// TwinCAT 3 PLC project Application
// ProgramVersion: 3.1.4024.0
// libraries:
//   Tc2_Standard, * (Beckhoff Automation GmbH)
//   Tc2_System, * (Beckhoff Automation GmbH)
//   Tc3_Module, * (Beckhoff Automation GmbH)
//   VisuDialogs, * (System)
//   VisuSymbols,3.5.10.0,System
// project tree:
//   DUTs/01_Schnittstellen/ I_HKSystem.TcIO (not stored), I_Magnetventil.TcIO (not stored), I_Motor1R.TcIO (not stored), I_Motor2R.TcIO, I_Sensor.TcIO
//   DUTs/02_Strukturen/ RezeptControlWord.TcDUT, RezeptStatusWord.TcDUT, SekControlWord.TcDUT, SystemStatusWord.TcDUT (not stored)
//   / GlobalTextList.TcGTLO, PlcTask.TcTTO, Visualisierungsmanager.TcVMO (not stored)
//   GVLs/01_OPC_UA/ GVL_OPC_UA.TcGVL
//   GVLs/ GVL.TcGVL
//   POUs/01_Objektklassen/ FB_A_HKSystem.TcPOU, FB_A_Magnetventil.TcPOU, FB_A_Motor1R.TcPOU, FB_A_Motor2R.TcPOU, FB_S_Sensor.TcPOU (not stored)
//   POUs/02_Anlage/01_Hilfsbausteine/ FB_Modus.TcPOU (not stored)
//   POUs/02_Anlage/ Reaktoreinheit.TcPOU
//   POUs/03_Grundfuntkionen/01_Vererbung/ FB_Basis.TcPOU
//   POUs/03_Grundfuntkionen/ GF_Befuellen.TcPOU, GF_Entleeren.TcPOU, GF_Pumpen.TcPOU, GF_Zirkulieren.TcPOU, GF_Ruehren.TcPOU, GF_Warten.TcPOU
//   POUs/04_Kommunikation/01_Hilfsfunktionsblock/ FB_Leitungswahl.TcPOU (not stored)
//   POUs/04_Kommunikation/ FB_Auswertung.TcPOU, Kommunikation.TcPOU
//   POUs/05_Simulation/ FB_SIM_Fuellstand.TcPOU
//   POUs/ MAIN.TcPOU
// real-time tasks:
//   TASK PlcTask: cycle T#10ms, priority 20, ADS port 350
//   TASK VISU_TASK: cycle T#200000us, priority 30, ADS port 351

CONFIGURATION Application
    RESOURCE PLC ON TwinCAT3
        TASK PlcTask(INTERVAL := T#10ms, PRIORITY := 20);
        PROGRAM MAIN WITH PlcTask : MAIN;
    END_RESOURCE
END_CONFIGURATION

// ---- DUTs/02_Strukturen/RezeptControlWord.TcDUT
TYPE RezeptControlWord :
STRUCT
	PowerOn			:BOOL;			// Einschalten von Reaktoreinheit
	SekReakt		:INT;			// Definierter sekundär-Reaktor
	Leitung			:INT;			// Definiert welche Leitung verwendet wird
	Temp			:REAL;			// Definierte Temperatur für Heiz- / Kühlprozess
	Enlteermenge	:REAL;			// Zu entleerende Menge
	Pumpmenge		:REAL;			// Zu pumpende Menge
	Haltedauer		:INT;			// Wie lange soll TEmperatur gehalten werden
	Ruehrdauer		:INT;			// Wie lange soll gerührt werden 
	Wartedauer		:INT;			// Wie lange soll gerührt werden
	Zirkulierdauer	:INT;			// Wie lange soll zirkuliert werden
END_STRUCT
END_TYPE

// ---- DUTs/02_Strukturen/RezeptStatusWord.TcDUT
TYPE RezeptStatusWord :
STRUCT
	SysReady		:BOOL;		// System ist bereit für Kommunikation
	SysActiv		:BOOL;		// System ist eingeschalten
	ReactReady		:BOOL;		// Primärreaktor ist bereit für den Prozess
	ReactActiv		:BOOL;		// Primärreaktor führt Prozess aus
	GF1Activ		:BOOL;		// Heiz- / Kühlprozess läuft
	GF2Activ		:BOOL;		// Entleerprozess läuft
	GF3Activ		:BOOL;		// Pumpprozess läuft
	GF4Activ		:BOOL;		// Halteprozess läuft
	GF5Activ		:BOOL;		// Rührprozess läuft
	GF6Activ		:BOOL;		// Warteprozess läuft
	GF7Activ		:BOOL;		// Auffüllprozess läuft
	GF8Activ		:BOOL;		// Zirkulierprozess läuft
END_STRUCT
END_TYPE

// ---- DUTs/02_Strukturen/SekControlWord.TcDUT
TYPE SekControlWord :
STRUCT
	// Das SekControlWord startet den Befüllprozess beim Sekundärreaktor (Empfänger)	
	R1				:BOOL;
	R2				:BOOL;
	R3				:BOOL;
	R4				:BOOL;
	R5				:BOOL;
	R6				:BOOL;
	R7				:BOOL;
END_STRUCT
END_TYPE

// ---- GVLs/01_OPC_UA/GVL_OPC_UA.TcGVL
{attribute 'qualified_only'}
VAR_GLOBAL
	// Rezept-Controlword
	{attribute 'OPC.UA.DA' := '1'}
	{attribute 'OPC.UA.DA.StructuredType' := '1'}
	CW			:RezeptControlWord;
	
	// Rezept-Statusword
	{attribute 'OPC.UA.DA' := '1'}
	{attribute 'OPC.UA.DA.Access' := '1'}
	{attribute 'OPC.UA.DA.StructuredType' := '1'}
	SW			:RezeptStatusWord;
	
	// System-Statusword
	{attribute 'OPC.UA.DA' := '1'}
	{attribute 'OPC.UA.DA.StructuredType' := '1'}
	SysSW		:SystemStatusWord;
	
	// Sekundärreaktor-Controlword
	{attribute 'OPC.UA.DA' := '1'}
	{attribute 'OPC.UA.DA.StructuredType' := '1'}
	SekCW		:SekControlWord;
END_VAR

// ---- GVLs/GVL.TcGVL
{attribute 'qualified_only'}
VAR_GLOBAL
	
	// Systemzustand
	SysState			:INT;		// 0 = Grundfunktion nicht aktive | 1 = Grundfunktion aktive

	// Bedienparameter
	Bedien_Power		:BOOL;
	Bedien_Reset		:BOOL;
	
	// Debug-Variablen: 
	Debug_Verbunden		:BOOL := TRUE;
	Debug_Start			:BOOL := TRUE;
	Debug_SekStart		:BOOL;
	
	// Simulationsvariablen 
	Sim_StandSignal		:INT;
	Sim_Fuellen			:BOOL;

END_VAR

// ---- DUTs/01_Schnittstellen/I_Motor2R.TcIO
INTERFACE I_Motor2R

METHOD M_A_BWD : BOOL
VAR_INPUT
END_VAR
END_METHOD

METHOD M_A_FWD : BOOL
VAR_INPUT
END_VAR
END_METHOD

METHOD M_A_START : BOOL
VAR_INPUT
END_VAR
END_METHOD

METHOD M_A_STOP : BOOL
VAR_INPUT
END_VAR
END_METHOD

METHOD M_M_BWD : BOOL
VAR_INPUT
END_VAR
END_METHOD

METHOD M_M_FWD : BOOL
VAR_INPUT
END_VAR
END_METHOD

METHOD M_M_START : BOOL
VAR_INPUT
END_VAR
END_METHOD

METHOD M_M_STOP : BOOL
VAR_INPUT
END_VAR
END_METHOD

PROPERTY P_Laufzeit : TIME
GET
END_GET
END_PROPERTY

PROPERTY P_MaxDrz : INT
SET
END_SET
END_PROPERTY

PROPERTY P_Status : INT
GET
END_GET
END_PROPERTY

END_INTERFACE

// ---- DUTs/01_Schnittstellen/I_Sensor.TcIO
INTERFACE I_Sensor

PROPERTY P_GrenzeOben : BOOL
GET
END_GET
END_PROPERTY

PROPERTY P_GrenzeUnten : BOOL
GET
END_GET
END_PROPERTY

PROPERTY P_Messwert : REAL
GET
END_GET
END_PROPERTY

END_INTERFACE

// ---- POUs/MAIN.TcPOU
PROGRAM MAIN
VAR
	Simulation		:FB_Sim_Fuellstand;
	Sim_ON			:BOOL := TRUE;
END_VAR

VAR_INPUT
	// Statusword
	
	// Sonstiges
END_VAR

// Starten der Reaktoreinheit
Reaktoreinheit();

// Starten der Auswertung der Kommunikationsschnittstelle
Kommunikation();

// Simulation starten
IF Sim_ON THEN
	Simulation(I_Fuellen := GVL.Sim_Fuellen,
			   O_SensorSignal => GVL.Sim_StandSignal);
			   
	Reaktoreinheit.F1.I_iSignal := GVL.Sim_StandSignal;
END_IF

END_PROGRAM

// ---- POUs/05_Simulation/FB_SIM_Fuellstand.TcPOU
FUNCTION_BLOCK FB_SIM_Fuellstand
VAR_INPUT
	I_Fuellen			:BOOL;
END_VAR

VAR_OUTPUT
	O_SensorSignal		:INT;
END_VAR
	
VAR
	V_Delay				:TON;
	V_TimeStatus		:BOOL;
END_VAR

// Timer instanziieren
V_Delay(IN := V_TimeStatus, PT := T#1S);	

IF I_Fuellen THEN
	// Grundwert definieren
	O_SensorSignal := 0;
	
	// Timer starten
	V_TimeStatus := TRUE;
	
	// Reaktor füllen
	IF V_Delay.Q THEN
		V_TimeStatus := FALSE;
		O_SensorSignal := O_SensorSignal + (27648/100);
	END_IF
END_IF

END_FUNCTION_BLOCK

// ---- POUs/02_Anlage/Reaktoreinheit.TcPOU
PROGRAM Reaktoreinheit
VAR
	// Allgemeine Instanziierungen
	Mode					:FB_Modus;
	
	// Instanziierung der Aktoren
	YSE1, YSE2				:FB_A_Magnetventil;
	YSA1, YSA2, YSA3		:FB_A_Magnetventil;
	YSP1, YSP2, YSP3		:FB_A_Magnetventil;
	
	NC1						:FB_A_Motor1R;
	
	PS1						:FB_A_Motor2R;
	
	HKP1					:FB_A_HKSystem;
END_VAR

VAR_INPUT
		// Instanziierung der Sensoren
	T1						:FB_S_Sensor;
	F1						:FB_S_Sensor;
END_VAR

YSE1(I_iModus := Mode.O_iModus); // FB_A_Magnetventil
YSP3(I_iModus := Mode.O_iModus); // FB_A_Magnetventil
F1(I_rHigh := 27648, I_rLow := 0, I_rMax := 100, I_rMin := 0); // FB_S_Sensor
Mode(I_bPower := GVL.Bedien_Power); // FB_Modus
YSA3(I_iModus := Mode.O_iModus); // FB_A_Magnetventil
HKP1(
    I_bVerbunden := GVL.Debug_Verbunden,
    I_iModus := Mode.O_iModus,
    I_iTemp := T1.P_Messwert,
    I_bReset := GVL.Bedien_Reset); // FB_A_HKSystem
YSA2(I_iModus := Mode.O_iModus); // FB_A_Magnetventil
YSP2(I_iModus := Mode.O_iModus); // FB_A_Magnetventil
PS1(
    I_bVerbunden := GVL.Debug_Verbunden,
    I_iModus := Mode.O_iModus,
    I_bReset := GVL.Bedien_Reset,
    I_iGeschw := 100); // FB_A_Motor2R
NC1(I_iModus := Mode.O_iModus, I_bReset := GVL.Bedien_Reset, I_iGeschw := 100); // FB_A_Motor1R
YSE2(I_iModus := Mode.O_iModus); // FB_A_Magnetventil
YSA1(I_iModus := Mode.O_iModus); // FB_A_Magnetventil
YSP1(I_iModus := Mode.O_iModus); // FB_A_Magnetventil
T1(I_rHigh := 27648, I_rLow := 0, I_rMax := 100, I_rMin := 0); // FB_S_Sensor

END_PROGRAM

// ---- POUs/01_Objektklassen/FB_A_Magnetventil.TcPOU
FUNCTION_BLOCK FB_A_Magnetventil IMPLEMENTS I_Magnetventil
VAR_INPUT
	I_iModus			:INT;		// Zustand des Systems (z.B. 0 = AUS | 1 = MAN | 2 = AUTO)
	I_bVerriegeln		:BOOL;		// Verriegelte Elemente sind nicht ansteuerbar
END_VAR

VAR_OUTPUT
	O_bAktivieren		:BOOL;		// Ventil wird geöffnet / geschlossen
	O_bStoerung			:BOOL;		// Befindet sich das Element in einem Error
	O_iStoerungID		:INT;		// Anzeigen von Störung über eine INT-Variable
END_VAR

VAR
END_VAR

// Verriegeln des Systems (Element geht in definierten Zustand) -> Ventil wird geschlossen
IF I_bVerriegeln THEN
	O_bAktivieren := FALSE;
END_IF

METHOD M_A_OEFFNEN : BOOL
VAR_INPUT
END_VAR
// EBENE 1: Verriegelung
IF NOT I_bVerriegeln THEN	
	// EBEN 2: AUTO-Modus
		IF I_iModus = 2 THEN
			O_bAktivieren := TRUE;
		END_IF
END_IF

M_A_OEFFNEN := O_bAktivieren;
END_METHOD

METHOD M_A_SCHLIESSEN : BOOL
VAR_INPUT
END_VAR
IF I_iModus = 2 THEN
	O_bAktivieren := FALSE;
END_IF

M_A_SCHLIESSEN := NOT O_bAktivieren;
END_METHOD

METHOD M_M_OEFFNEN : BOOL
VAR_INPUT
END_VAR
// EBENE 1: Verriegelung
IF NOT I_bVerriegeln THEN	
	// EBEN 2: MAN-Modus
		IF I_iModus = 1 THEN
			O_bAktivieren := TRUE;
		END_IF
END_IF

M_M_OEFFNEN := O_bAktivieren;
END_METHOD

METHOD M_M_SCHLIESSEN : BOOL
VAR_INPUT
END_VAR
IF I_iModus = 1 THEN
	O_bAktivieren := FALSE;
END_IF

M_M_SCHLIESSEN := NOT O_bAktivieren;
END_METHOD

PROPERTY P_Status : INT
GET
IF O_bAktivieren THEN
	P_Status := 1;
ELSE
	P_Status := 0;
END_IF

IF I_bVerriegeln THEN
	P_Status := 10;
END_IF
END_GET
END_PROPERTY

END_FUNCTION_BLOCK

// ---- POUs/01_Objektklassen/FB_A_Motor1R.TcPOU
FUNCTION_BLOCK FB_A_Motor1R IMPLEMENTS I_Motor1R
VAR_INPUT
	I_iModus			:INT;		// Zustand des Systems (z.B. 0 = AUS | 1 = MAN | 2 = AUTO | 3 = Error)
	I_bVerriegeln		:BOOL;		// Verriegelte Elemente sind nicht ansteuerbar
	I_bReset			:BOOL;		// Zustand des Baustein wird zurückgesetzt 
	I_iGeschw			:INT;		// Angabe über Soll-Geschwindigkeit
END_VAR

VAR_OUTPUT
	O_bPower			:BOOL;		// Relais wird geschalten um FU mit Spannung zu versorgen
	O_iDrz				:INT;		// Ausgabe der Drehzahl für den Motor (Umrechnen von Spannung zu Drz)
	O_bStoerung			:BOOL;		// Befindet sich das Element in einem Error
	O_iStoerungID		:INT;		// Anzeigen von Störung über eine INT-Variable
END_VAR

VAR
	V_DrzMax		:INT;		// Variable für internes handling der Eigenschaft 
	V_Zeit			:TIME;		// Variable für internes handling der Eigenschaft 
	V_Status		:INT;		// Variable für internes handling der Eigenschaft 
	
	V_Timer			:TON;		// Runtime des Bausteins ermitteln
	
END_VAR

// Setzen der internen Variablen
P_MaxDrz := V_DrzMax;
V_Zeit := P_Laufzeit;
V_Status := P_Status;

// Reset des Bausteins
IF I_bReset THEN
	O_bStoerung := FALSE;
	O_iStoerungID := 0;
END_IF

// Verriegeln des Systems (Element geht in definierten Zustand) -> Motor wird gestoppt und ausgeschalten
IF I_bVerriegeln THEN
	O_iDrz := 0;
	O_bPower := FALSE;
END_IF

METHOD M_A_AN : BOOL
VAR_INPUT
END_VAR
// EBENE 1: Verriegelung
IF NOT I_bVerriegeln THEN	
	// EBEN 2: AUTO-Modus
		IF I_iModus = 2 THEN
			O_bPower := TRUE;
		END_IF
ELSE 
	O_bPower := FALSE;
END_IF

M_A_AN := O_bPower;
END_METHOD

METHOD M_A_AUS : BOOL
VAR_INPUT
END_VAR
IF I_iModus = 2 THEN
	O_bPower := FALSE;
	O_iDrz := 0;
END_IF

M_A_AUS := NOT O_bPower;
END_METHOD

METHOD M_A_START : BOOL
VAR_INPUT
END_VAR
// EBENE 1: Verriegelung
IF NOT I_bVerriegeln THEN

	// EBENE 2: Check der Drehzzahl
	IF I_iGeschw <= V_DrzMax THEN
		
		// Ebene 3: AUTO-Modus
		IF I_iModus = 2 THEN
			
			// EBENE 4: System muss AN sein
			IF O_bPower THEN
				O_iDrz := I_iGeschw;
				
			ELSE 	// Error: System ist nicht eingeschalten
				O_bStoerung := 1;
				O_iStoerungID := 11; 
		END_IF
		
	ELSE	// Error: Geschwindigkeit überschreitet die MaxDrz
		O_bStoerung := 1;
		O_iStoerungID := 12;
		END_IF		
	END_IF
END_IF

IF O_iDrz = I_iGeschw THEN
	M_A_START := TRUE;
ELSE
	M_A_START := FALSE;
END_IF
END_METHOD

METHOD M_A_STOP : BOOL
VAR_INPUT
END_VAR
// EBENE 1: Verriegelung
IF NOT I_bVerriegeln THEN
	O_iDrz := 0;
END_IF

IF O_iDrz = 0 THEN
	M_A_STOP := TRUE;
ELSE
	M_A_STOP := FALSE;
END_IF
END_METHOD

METHOD M_M_AN : BOOL
VAR_INPUT
END_VAR
// EBENE 1: Verriegelung
IF NOT I_bVerriegeln THEN	
	// EBEN 2: MAN-Modus
		IF I_iModus = 1 THEN
			O_bPower := TRUE;
		END_IF
ELSE 
	O_bPower := FALSE;
END_IF

M_M_AN := O_bPower;
END_METHOD

METHOD M_M_AUS : BOOL
VAR_INPUT
END_VAR
IF I_iModus = 1 THEN
	O_bPower := FALSE;
	O_iDrz := 0;
END_IF

M_M_AUS := NOT O_bPower;
END_METHOD

METHOD M_M_START : BOOL
VAR_INPUT
END_VAR
// EBENE 1: Verriegelung
IF NOT I_bVerriegeln THEN

	// EBENE 2: Check der Drehzzahl
	IF I_iGeschw <= V_DrzMax THEN
		
		// EBENE 3: MAN-Modus
		IF I_iModus = 1 THEN
			
			// EBENE 4: System muss AN sein
			IF O_bPower THEN
				O_iDrz := I_iGeschw;
				
			ELSE 	// Error: System ist nicht eingeschalten
				O_bStoerung := 1;
			O_iStoerungID := 11;
			END_IF
		END_IF
		
	ELSE	// Error: Geschwindigkeit überschreitet die MaxDrz
		O_bStoerung := 1;
		O_iStoerungID := 12;
	END_IF		
END_IF

IF O_iDrz = I_iGeschw THEN
	M_M_START := TRUE;
ELSE
	M_M_START := FALSE;
END_IF
END_METHOD

METHOD M_M_STOP : BOOL
VAR_INPUT
END_VAR
// EBENE 1: Verriegelung
IF NOT I_bVerriegeln THEN
	O_iDrz := 0;
END_IF

IF O_iDrz = 0 THEN
	M_M_STOP := TRUE;
ELSE
	M_M_STOP := FALSE;
END_IF
END_METHOD

PROPERTY PUBLIC P_Laufzeit : TIME
GET
IF O_iDrz > 0 THEN
	V_Timer(IN := TRUE, PT := T#100H);
END_IF

IF O_iDrz = 0 THEN
	V_Timer(IN := FALSE);
END_IF 
P_Laufzeit := V_Timer.ET;
END_GET
END_PROPERTY

PROPERTY PUBLIC P_MaxDrz : INT
SET
END_SET
END_PROPERTY

PROPERTY PUBLIC P_Status : INT
GET
IF O_bPower THEN
	P_Status := 1;
ELSE
	P_Status := 0;
END_IF

IF O_iDrz > 0 AND O_bPower THEN
	P_Status := 2;
END_IF

IF I_bVerriegeln THEN
	P_Status := 10;
END_IF
END_GET
END_PROPERTY

END_FUNCTION_BLOCK

// ---- POUs/01_Objektklassen/FB_A_Motor2R.TcPOU
FUNCTION_BLOCK FB_A_Motor2R IMPLEMENTS I_Motor2R
VAR_INPUT
	I_bVerbunden		:BOOL;		// Angabe ob Pumpe angeschlossen ist
	I_iModus			:INT;		// Zustand des Systems (z.B. 0 = AUS | 1 = MAN | 2 = AUTO)
	I_bVerriegeln		:BOOL;		// Verriegelte Elemente sind nicht ansteuerbar
	I_bReset			:BOOL;		// Zustand des Baustein wird zurückgesetzt 
	I_iGeschw			:INT;		// Angabe über Soll-Geschwindigkeit
END_VAR

VAR_OUTPUT
	
	O_iDrz				:INT;		// Ausgabe der Drehzahl für den Motor
	O_bRichtung			:BOOL;		// Ausgabe der Drehrichtung
	O_bStoerung			:BOOL;		// Befindet sich das Element in einem Error
	O_iStoerungID		:INT;		// Anzeigen von Störung über eine INT-Variable
END_VAR

VAR
	V_DrzMax		:INT;		// Variable für internes handling der Eigenschaft 
	V_Zeit			:TIME;		// Variable für internes handling der Eigenschaft 
	V_Zustand		:INT;		// Variable für internes handling der Eigenschaft

	V_Timer			:TON;		// Runtime des Bausteins ermitteln 
END_VAR

// Setzen der internen Variablen
P_MaxDrz := V_DrzMax;
V_Zeit := P_Laufzeit;
V_Zustand := P_Status;

// Reset des Bausteins
IF I_bReset THEN
	O_bStoerung := FALSE;
	O_iStoerungID := 0;
END_IF

// Verriegeln des Systems (Element geht in definierten Zustand) -> Motor wird hält an 
IF I_bVerriegeln THEN
	O_iDrz := 0;
	O_bRichtung := FALSE;
END_IF

METHOD M_A_BWD : BOOL
VAR_INPUT
END_VAR
// EBENE 1: Verriegelung
IF NOT I_bVerriegeln THEN	
	// EBENE 2: AUTO-Modus
		IF I_iModus = 2 THEN
			// EBENE 3: System muss angeschlossen sein
			IF I_bVerbunden THEN
				O_bRichtung := TRUE;
			ELSE 	// Error: System ist nicht angeschlossen
				O_bStoerung := 1;
				O_iStoerungID := 03;
			END_IF
		END_IF
END_IF

M_A_BWD := O_bRichtung;
END_METHOD

METHOD M_A_FWD : BOOL
VAR_INPUT
END_VAR
// EBENE 1: Verriegelung
IF NOT I_bVerriegeln THEN	
	// EBENE 2: AUTO-Modus
		IF I_iModus = 2 THEN
			// EBENE 3: System muss angeschlossen sein
			IF I_bVerbunden THEN
				O_bRichtung := FALSE;
			ELSE 	// Error: System ist nicht angeschlossen
				O_bStoerung := 1;
				O_iStoerungID := 03;
			END_IF
		END_IF
END_IF

M_A_FWD := NOT O_bRichtung;
END_METHOD

METHOD M_A_START : BOOL
VAR_INPUT
END_VAR
// EBENE 1: Verriegelung
IF NOT I_bVerriegeln THEN

	// EBENE 2: Check der Drehzzahl
	IF I_iGeschw <= V_DrzMax THEN
		
		// EBENE 3: AUTO-Modus
		IF I_iModus = 2 THEN
			
			// EBENE 4: System muss angeschlossen sein
			IF I_bVerbunden THEN
				O_iDrz := I_iGeschw;
				
			ELSE 	// Error: System ist nicht angeschlossen
				O_bStoerung := 1;
				O_iStoerungID := 03;
			END_IF
		END_IF
		
	ELSE	// Error: Geschwindigkeit überschreitet die MaxDrz
		O_bStoerung := 1;
		O_iStoerungID := 01;
	END_IF		
END_IF

IF O_iDrz = I_iGeschw THEN
	M_A_START := TRUE;
END_IF
END_METHOD

METHOD M_A_STOP : BOOL
VAR_INPUT
END_VAR
// EBENE 1: Verriegelung
IF NOT I_bVerriegeln THEN
	O_iDrz := 0;
END_IF

IF O_iDrz = 0 THEN
	M_A_STOP := TRUE;
END_IF
END_METHOD

METHOD M_M_BWD : BOOL
VAR_INPUT
END_VAR
// EBENE 1: Verriegelung
IF NOT I_bVerriegeln THEN	
	// EBENE 2: MAN-Modus
		IF I_iModus = 1 THEN
			// EBENE 3: System muss angeschlossen sein
			IF I_bVerbunden THEN
				O_bRichtung := TRUE;
			ELSE 	// Error: System ist nicht angeschlossen
				O_bStoerung := 1;
				O_iStoerungID := 03;
			END_IF
		END_IF
END_IF

M_M_BWD := O_bRichtung;
END_METHOD

METHOD M_M_FWD : BOOL
VAR_INPUT
END_VAR
// EBENE 1: Verriegelung
IF NOT I_bVerriegeln THEN	
	// EBENE 2: MAN-Modus
		IF I_iModus = 1 THEN
			// EBENE 3: System muss angeschlossen sein
			IF I_bVerbunden THEN
				O_bRichtung := FALSE;
			ELSE 	// Error: System ist nicht angeschlossen
				O_bStoerung := 1;
				O_iStoerungID := 03;
			END_IF
		END_IF
END_IF

M_M_FWD := NOT O_bRichtung;
END_METHOD

METHOD M_M_START : BOOL
VAR_INPUT
END_VAR
// EBENE 1: Verriegelung
IF NOT I_bVerriegeln THEN

	// EBENE 2: Check der Drehzzahl
	IF I_iGeschw <= V_DrzMax THEN
		
		// EBENE 3: MAN-Modus
		IF I_iModus = 1 THEN
			
			// EBENE 4: System muss angeschlossen sein
			IF I_bVerbunden THEN
				O_iDrz := I_iGeschw;
				
			ELSE 	// Error: System ist nicht angeschlossen
				O_bStoerung := 1;
				O_iStoerungID := 03;
			END_IF
		END_IF
		
	ELSE	// Error: Geschwindigkeit überschreitet die MaxDrz
		O_bStoerung := 1;
		O_iStoerungID := 01;
	END_IF		
END_IF

IF O_iDrz = I_iGeschw THEN
	M_M_START := TRUE;
END_IF
END_METHOD

METHOD M_M_STOP : BOOL
VAR_INPUT
END_VAR
// EBENE 1: Verriegelung
IF NOT I_bVerriegeln THEN
	O_iDrz := 0;
END_IF

IF O_iDrz = 0 THEN
	M_M_STOP := TRUE;
END_IF
END_METHOD

PROPERTY PUBLIC P_Laufzeit : TIME
GET
IF O_iDrz > 0 THEN
	V_Timer(IN := TRUE, PT := T#100H);
END_IF

IF O_iDrz = 0 THEN
	V_Timer(IN := FALSE);
END_IF 
P_Laufzeit := V_Timer.ET;
END_GET
END_PROPERTY

PROPERTY PUBLIC P_MaxDrz : INT
SET
END_SET
END_PROPERTY

PROPERTY PUBLIC P_Status : INT
GET
IF I_bVerbunden THEN
	P_Status := 1;
END_IF

IF I_bVerriegeln THEN
	P_Status := 10;
END_IF

IF O_iDrz > 0	THEN
	P_Status := 2;
END_IF
END_GET
END_PROPERTY

END_FUNCTION_BLOCK

// ---- POUs/01_Objektklassen/FB_A_HKSystem.TcPOU
FUNCTION_BLOCK FB_A_HKSystem IMPLEMENTS I_HKSystem
VAR_INPUT
	I_bVerbunden	:BOOL;		// Angabe ob HK-System angeschlossen ist
	I_iModus		:INT;		// Zustand des Systems (z.B. 0 = AUS | 1 = MAN | 2 = AUTO)
	I_iTemp			:REAL;		// Aktuelle Temperatur um Heizmodus auszuwählen und zu stoppen
	I_bVerriegeln	:BOOL;		// Verriegelte Elemente sind nicht ansteuerbar
	I_bReset		:BOOL;		// Zustand des Baustein wird zurückgesetzt 
END_VAR

VAR_OUTPUT
	O_bPumpen		:BOOL;		// Pumpe des HK-Systems wird betrieben
	O_bKuehlen		:BOOL;		// HK-System heizt das Medium auf
	O_bHeizen		:BOOL;		// HK-System kühlt das Medium ab
	O_bStoerung		:BOOL;		// Befindet sich das Element in einem Error
	O_iStoerungID	:INT;		// Anzeigen von Störung über eine INT-Variable
	
END_VAR
	
VAR
	V_DefTemp		:INT;		// Variable für internes handling der Eigenschaft 
	V_Zeit			:TIME;		// Variable für internes handling der Eigenschaft 
	V_Zustand		:INT;		// Variable für internes handling der Eigenschaft 
	
	V_Timer			:TON;		// Runtime des Bausteins ermitteln
END_VAR

// Setzen der internen Variablen
V_Zeit := P_Laufzeit;
V_Zustand := P_Zustand;

// Fehler durch Verbindungsabbruch
IF O_bPumpen OR O_bKuehlen OR O_bHeizen THEN
	IF NOT I_bVerbunden THEN
		O_bPumpen := FALSE;
		O_bKuehlen := FALSE;
		O_bHeizen := FALSE;
		
		O_bStoerung := TRUE;
		O_iStoerungID := 04;
	END_IF
END_IF

// Abbruch des Heiz-Kühlprozesses beim erreichen der Temp
IF O_bHeizen OR O_bKuehlen THEN 
	IF I_iTemp = V_DefTemp THEN
		O_bKuehlen := FALSE;
		O_bHeizen := FALSE;		
	END_IF
END_IF

// Reset des Bausteins
IF I_bReset THEN
	O_bStoerung := FALSE;
	O_iStoerungID := 0;
END_IF

METHOD M_A_HK_AN : BOOL
VAR_INPUT
END_VAR
// EBENE 1: Verriegelung
IF NOT I_bVerriegeln THEN	
	// EBENE 2: AUTO-Modus
		IF I_iModus = 2 THEN
			// EBENE 3: Ist Pumpe AN
				IF O_bPumpen THEN
				// EBENE 4: Heizen oder Kühlen
					IF V_DefTemp > I_iTemp THEN
						O_bKuehlen := FALSE;
						O_bHeizen := TRUE;
						
						M_A_HK_AN := O_bHeizen;
						
					ELSIF I_iTemp > V_DefTemp THEN 	
						O_bHeizen := FALSE;
						O_bKuehlen := TRUE;
						
						M_A_HK_AN := O_bKuehlen;
					END_IF
				ELSE // Error: System ist nicht eingeschalten
					O_bStoerung := 1;
					O_iStoerungID := 11; 
				END_IF
			END_IF
END_IF
END_METHOD

METHOD M_A_HK_AUS : BOOL
VAR_INPUT
END_VAR
// EBENE 1: Verriegelung
IF NOT I_bVerriegeln THEN
		O_bKuehlen := FALSE;
		O_bHeizen := FALSE;
END_IF

IF O_bKuehlen = FALSE THEN
	M_A_HK_AUS := TRUE;
END_IF
END_METHOD

METHOD M_A_PUMPE_AN : BOOL
VAR_INPUT
END_VAR
// EBENE 1: Verriegelung
IF NOT I_bVerriegeln THEN	
	// EBENE 2: AUTO-Modus
		IF I_iModus = 2 THEN
			// EBENE 3: System muss angeschlossen sein
			IF I_bVerbunden THEN
				O_bPumpen := TRUE;
			ELSE 	// Error: System ist nicht angeschlossen
				O_bStoerung := 1;
				O_iStoerungID := 03;
			END_IF
		END_IF
END_IF

M_A_PUMPE_AN := O_bPumpen;
END_METHOD

METHOD M_A_PUMPE_AUS : BOOL
VAR_INPUT
END_VAR
// EBENE 1: Verriegelung
IF NOT I_bVerriegeln THEN
	IF NOT O_bHeizen AND NOT O_bKuehlen THEN
		O_bPumpen := FALSE;
	ELSE
		O_bStoerung := TRUE;
		O_iStoerungID := 05;
	END_IF
END_IF

IF O_bPumpen = FALSE THEN
	M_A_PUMPE_AUS := TRUE;
END_IF
END_METHOD

METHOD M_M_HK_AN : BOOL
VAR_INPUT
END_VAR
// EBENE 1: Verriegelung
IF NOT I_bVerriegeln THEN	
	// EBENE 2: MAN-Modus
		IF I_iModus = 1 THEN
			// EBENE 3: Ist Pumpe AN
				IF O_bPumpen THEN
				// EBENE 4: Heizen oder Kühlen
					IF V_DefTemp > I_iTemp THEN
						O_bKuehlen := FALSE;
						O_bHeizen := TRUE;
						
						M_M_HK_AN := O_bHeizen;
						
					ELSIF I_iTemp > V_DefTemp THEN 	
						O_bHeizen := FALSE;
						O_bKuehlen := TRUE;
						
						M_M_HK_AN := O_bKuehlen;
					END_IF
				ELSE // Error: System ist nicht eingeschalten
				O_bStoerung := 1;
				O_iStoerungID := 11; 	
				END_IF
			END_IF
END_IF
END_METHOD

METHOD M_M_HK_AUS : BOOL
VAR_INPUT
END_VAR
// EBENE 1: Verriegelung
IF NOT I_bVerriegeln THEN
		O_bKuehlen := FALSE;
		O_bHeizen := FALSE;
END_IF

IF O_bKuehlen = FALSE THEN
	M_M_HK_AUS := TRUE;
END_IF
END_METHOD

METHOD M_M_PUMPE_AN : BOOL
VAR_INPUT
END_VAR
// EBENE 1: Verriegelung
IF NOT I_bVerriegeln THEN	
	// EBENE 2: MAN-Modus
		IF I_iModus = 1 THEN
			// EBENE 3: System muss angeschlossen sein
			IF I_bVerbunden THEN
				O_bPumpen := TRUE;
			ELSE 	// Error: System ist nicht angeschlossen
				O_bStoerung := 1;
				O_iStoerungID := 03;
			END_IF
		END_IF
END_IF

M_M_PUMPE_AN := O_bPumpen;
END_METHOD

METHOD M_M_PUMPE_AUS : BOOL
VAR_INPUT
END_VAR
// EBENE 1: Verriegelung
IF NOT I_bVerriegeln THEN
	IF NOT O_bHeizen AND NOT O_bKuehlen THEN
		O_bPumpen := FALSE;
	ELSE
		O_bStoerung := TRUE;
		O_iStoerungID := 05;
	END_IF
END_IF

IF O_bPumpen = FALSE THEN
	M_M_PUMPE_AUS := TRUE;
END_IF
END_METHOD

PROPERTY P_DefTemp : INT
SET
END_SET
END_PROPERTY

PROPERTY P_Laufzeit : TIME
GET
IF O_bKuehlen OR O_bHeizen THEN
	V_Timer(IN := TRUE, PT := T#100H);
ELSE
	V_Timer(IN := FALSE);
END_IF

P_Laufzeit := V_Timer.ET;
END_GET
END_PROPERTY

PROPERTY PUBLIC P_Zustand : INT
GET
END_GET
END_PROPERTY

END_FUNCTION_BLOCK

// ---- POUs/04_Kommunikation/Kommunikation.TcPOU
PROGRAM Kommunikation
VAR
	
	// Instanziierung der Auswertung:
	Auswertung		:FB_Auswertung;
	Mode			:FB_Modus;
	
	// Instanziierung der Grundfunktionen: 
	Entleeren		:GF_Entleeren;
	//Halten			:GF_Halten;
	Pumpen			:GF_Pumpen;
	Zirkulieren		:GF_Zirkulieren;
	Ruehren 		:GF_Ruehren;
	Warten			:GF_Warten;	
	Befuellen		:GF_Befuellen;	
	Leitung			:FB_Leitungswahl;

END_VAR

Auswertung(
    I_RNr := GVL_OPC_UA.CW.SekReakt,
    I_ControlWord := GVL_OPC_UA.CW,
    I_SystemStatusWord := GVL_OPC_UA.SysSW,
    I_SekCW := GVL_OPC_UA.SekCW); // FB_Auswertung
GVL_OPC_UA.SW := Auswertung.O_StatusWord;
GVL.Bedien_Power := Auswertung.O_SystemON;

END_PROGRAM

// ---- POUs/04_Kommunikation/FB_Auswertung.TcPOU
FUNCTION_BLOCK FB_Auswertung
VAR_INPUT
	I_Manuel			:BOOL;	
	I_RNr				:INT;				// Reaktornummer für korrekte Zuweisung von SystemStatusWord		
	I_ControlWord		:RezeptControlWord;
	I_SystemStatusWord	:SystemStatusWord;
	I_SekCW				:SekControlWord;
END_VAR
VAR_OUTPUT
	O_StatusWord		:RezeptStatusWord; 
	O_SystemON			:BOOL;
END_VAR
VAR
	V_Status			:INT;						// Variable für Case-Switch
	V_Aktiv				:BOOL;						// System ist aktiv
	V_GF_Switch			:INT;						// Definiert welche GF durchgegührt werden soll	
	V_SekRe				:BOOL;						// Wird aktiviert falls Reaktor als Sekundärreaktor eingesetzt wird
	V_SekReady			:BOOL;
	V_SekActiv			:BOOL;
END_VAR

// Befindet sich System in Manuel-Modus
IF I_Manuel THEN
	V_Status := 0;
END_IF  

// System befindet sich im Automatik-Modus, aber ist noch nicht aktiv
IF NOT I_Manuel AND NOT V_Aktiv THEN
	V_Status := 1;
END_IF

// Auswertung des SystemStatusWords 
CASE I_RNr OF 
	1:	V_SekReady := I_SystemStatusWord.R1_Ready;
		V_SekActiv := I_SystemStatusWord.R1_Activ;
	
	2:	V_SekReady := I_SystemStatusWord.R2_Ready;
		V_SekActiv := I_SystemStatusWord.R2_Activ;
	
	3:	V_SekReady := I_SystemStatusWord.R3_Ready;
		V_SekActiv := I_SystemStatusWord.R3_Activ;
	
	4:	V_SekReady := I_SystemStatusWord.R4_Ready;
		V_SekActiv := I_SystemStatusWord.R4_Activ;
		
	5:	V_SekReady := I_SystemStatusWord.R5_Ready;
		V_SekActiv := I_SystemStatusWord.R5_Activ;
	
	6:	V_SekReady := I_SystemStatusWord.R6_Ready;
		V_SekActiv := I_SystemStatusWord.R6_Activ;
	
	7:	V_SekReady := I_SystemStatusWord.R7_Ready;
		V_SekActiv := I_SystemStatusWord.R7_Activ;
END_CASE

CASE V_Status OF
	0: // System im Manuel-Modus
		O_StatusWord.SysReady := FALSE;
		
	//==================================================================================================
	1: // Auswerten von Controlwords bezüglich Systemstart
		// System ist Ready für Communikation
		O_StatusWord.SysReady := TRUE;
		
		// Falls Power eingeschalten wird und das System noch nicht Ein ist, wird System Aktiviert
		IF I_ControlWord.PowerOn AND NOT O_SystemON THEN
			V_Aktiv := TRUE;
			V_Status := 2;
		END_IF
		
		// Auswertung von Sekundärreaktor-Controlword bezüglich Empfänger-Prozes 
		CASE I_RNr OF 
			1: V_SekRe := I_SekCW.R1;
			2: V_SekRe := I_SekCW.R2;
			3: V_SekRe := I_SekCW.R3;
			4: V_SekRe := I_SekCW.R4;
			5: V_SekRe := I_SekCW.R5;
			6: V_SekRe := I_SekCW.R6;
			7: V_SekRe := I_SekCW.R7;
		END_CASE
		
		IF V_SekRe THEN
			V_Aktiv := TRUE;
			V_Status := 2;
		END_IF
	
	//==================================================================================================
	2: // System wird eingeschaltet
			O_SystemON := TRUE;
			O_StatusWord.SysActiv := TRUE;
			
			IF GVL.Bedien_Power THEN
				V_Status := 3;
			END_IF
	//==================================================================================================
	3: // Leitung wird definiert
			
			V_Status := 4;
	//==================================================================================================
	4: // Prozess wird durchgeführt
		IF I_ControlWord.Enlteermenge > 0 THEN
			V_GF_Switch := 1;
			Kommunikation.Entleeren.M_START();
			V_Status := 5;
		END_IF
		
		IF I_ControlWord.Pumpmenge > 0 THEN
			V_GF_Switch := 2;
			Kommunikation.Pumpen.M_START();
			V_Status := 5;
		END_IF
		
		IF I_ControlWord.Haltedauer > 0 THEN
			V_GF_Switch := 3;
			V_Status := 5;
		END_IF
		
		IF I_ControlWord.Ruehrdauer > 0 THEN
			V_GF_Switch := 4;
			Kommunikation.Ruehren.M_START();
			V_Status := 5;
		END_IF
		
		IF I_ControlWord.Wartedauer > 0 THEN
			// Parameter, dass System zurückgesetzt wird (Start-Situation)
			// Damit können funktionen besser getestet werden
			IF I_ControlWord.Wartedauer = 99 THEN
				O_StatusWord.ReactReady := 0;
				O_StatusWord.ReactActiv := 0;
				O_StatusWord.GF1Activ := 0;
				O_StatusWord.GF2Activ := 0;
				O_StatusWord.GF3Activ := 0;
				O_StatusWord.GF4Activ := 0;
				O_StatusWord.GF5Activ := 0;
				O_StatusWord.GF6Activ := 0;
				O_StatusWord.GF7Activ := 0;
				O_StatusWord.GF8Activ := 0;
				V_Status := 6;
			ELSE 
				V_GF_Switch := 5;
				Kommunikation.Warten.M_START();
				V_Status := 5;
			END_IF
		END_IF
		
		IF I_ControlWord.Zirkulierdauer > 0 THEN
			V_GF_Switch := 6;
			Kommunikation.Zirkulieren.M_START();
			V_Status := 5;
		END_IF
		
		IF V_SekRe THEN
			V_GF_Switch := 7;
			Kommunikation.Befuellen.M_START();
			V_Status := 5;
		END_IF
		
	//==================================================================================================
	5: // System wartete auf Abschluss von Prozess
		CASE V_GF_Switch OF 
			1:	ACT_GF_Entleeren();
				IF Kommunikation.Entleeren.P_Status = 0 THEN
					V_Status := 6;
				END_IF
				
			2:	ACT_GF_Pumpen();
				IF Kommunikation.Pumpen.P_Status = 0 THEN
					V_Status := 6;
				END_IF
				
			3: //
			
			4:	ACT_GF_Ruehren();
				IF Kommunikation.Ruehren.P_Status = 0 THEN
					V_Status := 6;
				END_IF
				
			5:	ACT_GF_Warten();
				IF Kommunikation.Warten.P_Status = 0 THEN
					V_Status := 6;
				END_IF
				
			6:	ACT_GF_Zirkulieren();
				IF Kommunikation.Zirkulieren.P_Status = 0 THEN
					V_Status := 6;
				END_IF
				
			7: ACT_GF_Befuellen();
				IF Kommunikation.Befuellen.P_Status = 0 THEN
					V_Status := 6;
				END_IF
		END_CASE
	//==================================================================================================
	6: // System wird ausgeschalten
		IF NOT I_ControlWord.PowerOn THEN
			O_SystemON := FALSE;
			O_StatusWord.SysActiv := FALSE;
			V_Aktiv := FALSE; 
			V_Status := 1;
		END_IF
END_CASE

ACTION ACT_GF_Befuellen:
Kommunikation.Befuellen(
    I_Level := Reaktoreinheit.F1,
    I_Ventil := Kommunikation.Leitung.O_Ventil,
    I_CW := I_ControlWord); // GF_Befuellen
Kommunikation.Leitung(I_Ventil_1 := Reaktoreinheit.YSE1, I_Ventil_2 := Reaktoreinheit.YSE1); // FB_Leitungswahl
O_StatusWord := Kommunikation.Befuellen.O_SW;
END_ACTION

ACTION ACT_GF_Entleeren:
O_StatusWord := Kommunikation.Entleeren.O_SW;
Kommunikation.Entleeren(
    I_Level := Reaktoreinheit.F1,
    I_Ventil := Kommunikation.Leitung.O_Ventil,
    I_CW := I_ControlWord,
    I_SekReady := V_SekReady,
    I_SekActiv := V_SekActiv); // GF_Entleeren
Kommunikation.Leitung(I_Ventil_1 := Reaktoreinheit.YSA2, I_Ventil_2 := Reaktoreinheit.YSA3); // FB_Leitungswahl
END_ACTION

ACTION ACT_GF_Pumpen:
O_StatusWord := Kommunikation.Pumpen.O_SW;
Kommunikation.Pumpen(
    I_Ventil_IN := Reaktoreinheit.YSA1,
    I_Ventil_OUT := Kommunikation.Leitung.O_Ventil,
    I_Pumpe := Reaktoreinheit.PS1,
    I_CW := I_ControlWord,
    I_SekReady := V_SekReady,
    I_SekActiv := V_SekActiv); // GF_Pumpen
Kommunikation.Leitung(I_Ventil_1 := Reaktoreinheit.YSP1, I_Ventil_2 := Reaktoreinheit.YSP2); // FB_Leitungswahl
END_ACTION

ACTION ACT_GF_Ruehren:
O_StatusWord := Kommunikation.Ruehren.O_SW;
Kommunikation.Ruehren(I_Ruehrer := Reaktoreinheit.NC1, I_CW := I_ControlWord); // GF_Ruehren
END_ACTION

ACTION ACT_GF_Warten:
O_StatusWord := Kommunikation.Warten.O_SW;
Kommunikation.Warten(I_CW := I_ControlWord); // GF_Warten
END_ACTION

ACTION ACT_GF_Zirkulieren:
O_StatusWord := Kommunikation.Zirkulieren.O_SW;
Kommunikation.Zirkulieren(
    I_Ventil_IN := Reaktoreinheit.YSA1,
    I_Ventil_OUT := Reaktoreinheit.YSP3,
    I_Pumpe := Reaktoreinheit.PS1,
    I_CW := I_ControlWord); // GF_Zirkulieren
END_ACTION

END_FUNCTION_BLOCK

// ---- POUs/03_Grundfuntkionen/GF_Befuellen.TcPOU
FUNCTION_BLOCK GF_Befuellen	EXTENDS FB_Basis
VAR_INPUT
	// Instanzieren von Sensoren mit Interfaces
	I_Level		:I_Sensor;
	// Instanzieren von Aktoren mit Interfaces
	I_Ventil	:I_Magnetventil;
	// Rezeptparameter durch Controlword
	I_CW		:RezeptControlWord;	
END_VAR
VAR_OUTPUT
	O_SW		:RezeptStatusWord;
END_VAR
VAR
	
END_VAR

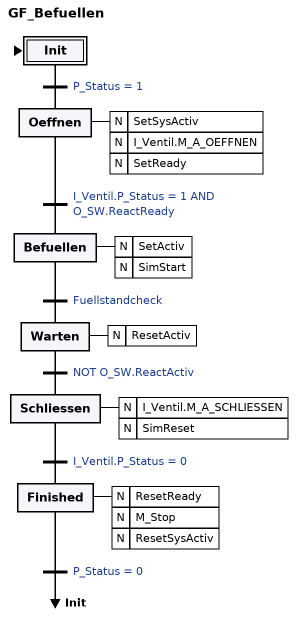
INITIAL_STEP Init:
END_STEP
TRANSITION FROM Init TO Oeffnen
    := P_Status = 1;
END_TRANSITION
STEP Oeffnen:
    SetSysActiv(N);
    I_Ventil.M_A_OEFFNEN(N);
    SetReady(N);
END_STEP
TRANSITION FROM Oeffnen TO Befuellen
    := I_Ventil.P_Status = 1 AND O_SW.ReactReady;
END_TRANSITION
STEP Befuellen:
    SetActiv(N);
    SimStart(N);
END_STEP
TRANSITION FROM Befuellen TO Warten
    := Fuellstandcheck;
END_TRANSITION
STEP Warten:
    ResetActiv(N);
END_STEP
TRANSITION FROM Warten TO Schliessen
    := NOT O_SW.ReactActiv;
END_TRANSITION
STEP Schliessen:
    I_Ventil.M_A_SCHLIESSEN(N);
    SimReset(N);
END_STEP
TRANSITION FROM Schliessen TO Finished_
    := I_Ventil.P_Status = 0;
END_TRANSITION
STEP Finished_:  // name as stored: Finished 
    ResetReady(N);
    M_Stop(N);
    ResetSysActiv(N);
END_STEP
TRANSITION FROM Finished_ TO Init
    := P_Status = 0;
END_TRANSITION

TRANSITION Fuellstandcheck:
// Prüfen welche Grundfunktion verwendet wird
IF I_CW.Enlteermenge > 0 THEN
	// Bedingung
	IF  I_CW.Enlteermenge < I_Level.P_Messwert THEN
		Fuellstandcheck := TRUE;
		
	ELSE 
		Fuellstandcheck := FALSE;
	END_IF
END_IF

// Prüfen welche Grundfunktion verwendet wird
IF I_CW.Pumpmenge > 0 THEN
	// Bedingung
	IF  I_CW.Pumpmenge < I_Level.P_Messwert THEN
		Fuellstandcheck := TRUE;
	ELSE 
		Fuellstandcheck := FALSE;
	END_IF
END_IF
END_TRANSITION

ACTION ResetActiv:
O_SW.ReactActiv := FALSE;
O_SW.GF7Activ := FALSE;
END_ACTION

ACTION ResetReady:
O_SW.ReactReady := FALSE;
END_ACTION

ACTION ResetSysActiv:
GVL.SysState := 0;
// Für Debug
GVL.Debug_SekStart := 0;
END_ACTION

ACTION SetActiv:
O_SW.ReactActiv := TRUE;
O_SW.GF7Activ := TRUE;
END_ACTION

ACTION SetReady:
O_SW.ReactReady := TRUE;
END_ACTION

ACTION SetSysActiv:
GVL.SysState := 1;
END_ACTION

ACTION SimReset:
GVL.Sim_Fuellen := FALSE;
END_ACTION

ACTION SimStart:
GVL.Sim_Fuellen := TRUE;
END_ACTION

END_FUNCTION_BLOCK

// ---- POUs/03_Grundfuntkionen/01_Vererbung/FB_Basis.TcPOU
FUNCTION_BLOCK FB_Basis
VAR_INPUT
END_VAR
VAR_OUTPUT
END_VAR
VAR
	V_Start			:BOOL;
END_VAR

METHOD M_START : BOOL
VAR_INPUT
END_VAR
V_Start := TRUE;
END_METHOD

METHOD M_STOP : BOOL
VAR_INPUT
END_VAR
V_Start := FALSE;
END_METHOD

PROPERTY P_Status : INT
GET
// 0 = Prozess läuft nicht
// 1 = Prozess läuft

IF V_Start THEN
	P_Status := 1;
ELSE
	P_Status := 0;
END_IF
END_GET
END_PROPERTY

END_FUNCTION_BLOCK

// ---- POUs/03_Grundfuntkionen/GF_Entleeren.TcPOU
FUNCTION_BLOCK GF_Entleeren	EXTENDS FB_Basis
VAR_INPUT
	// Instanzieren von Sensoren mit Interfaces
	I_Level			:I_Sensor;
	// Instanzieren von Aktoren mit Interfaces
	I_Ventil		:I_Magnetventil;
	// Rezeptparameter durch Controlword
	I_CW			:RezeptControlWord;
	I_SekReady		:BOOL;
	I_SekActiv		:BOOL;	
END_VAR
VAR_OUTPUT
	O_SW		:RezeptStatusWord;
END_VAR
VAR
	
END_VAR

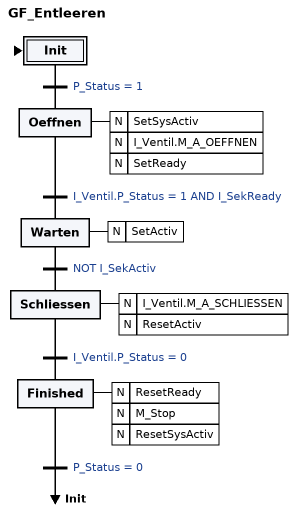
INITIAL_STEP Init:
END_STEP
TRANSITION FROM Init TO Oeffnen
    := P_Status = 1;
END_TRANSITION
STEP Oeffnen:
    SetSysActiv(N);
    I_Ventil.M_A_OEFFNEN(N);
    SetReady(N);
END_STEP
TRANSITION FROM Oeffnen TO Warten
    := I_Ventil.P_Status = 1 AND I_SekReady;
END_TRANSITION
STEP Warten:
    SetActiv(N);
END_STEP
TRANSITION FROM Warten TO Schliessen
    := NOT I_SekActiv;
END_TRANSITION
STEP Schliessen:
    I_Ventil.M_A_SCHLIESSEN(N);
    ResetActiv(N);
END_STEP
TRANSITION FROM Schliessen TO Finished
    := I_Ventil.P_Status = 0;
END_TRANSITION
STEP Finished:
    ResetReady(N);
    M_Stop(N);
    ResetSysActiv(N);
END_STEP
TRANSITION FROM Finished TO Init
    := P_Status = 0;
END_TRANSITION

ACTION ResetActiv:
O_SW.ReactActiv := FALSE;
O_SW.GF2Activ := FALSE;
END_ACTION

ACTION ResetReady:
O_SW.ReactReady := FALSE;
END_ACTION

ACTION ResetSysActiv:
GVL.SysState := 0;
END_ACTION

ACTION SetActiv:
O_SW.ReactActiv := TRUE;
O_SW.GF2Activ := TRUE;
END_ACTION

ACTION SetReady:
O_SW.ReactReady:= TRUE;
END_ACTION

ACTION SetSysActiv:
GVL.SysState := 1;
END_ACTION

END_FUNCTION_BLOCK

// ---- POUs/03_Grundfuntkionen/GF_Pumpen.TcPOU
FUNCTION_BLOCK GF_Pumpen EXTENDS FB_Basis
VAR_INPUT
	// Instanzieren von Sensoren mit Interfaces
	
	// Instanzieren von Aktoren mit Interfaces
	I_Ventil_IN		:I_Magnetventil;
	I_Ventil_OUT	:I_Magnetventil;
	
	I_Pumpe			:I_Motor2R;
	// Rezeptparameter durch Controlword
	I_CW			:RezeptControlWord;	
	I_SekReady		:BOOL;
	I_SekActiv		:BOOL;
END_VAR
VAR_OUTPUT
	O_SW		:RezeptStatusWord;
END_VAR
VAR
	
END_VAR

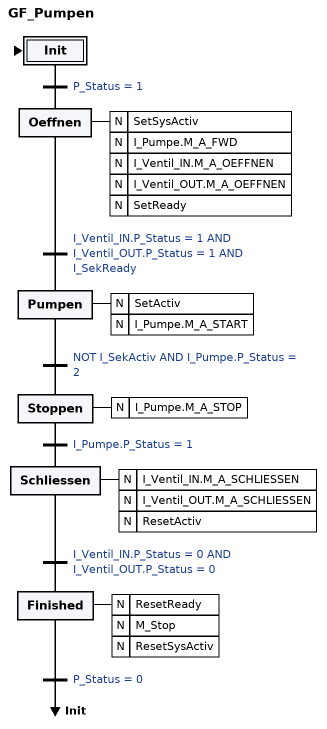
INITIAL_STEP Init:
END_STEP
TRANSITION FROM Init TO Oeffnen
    := P_Status = 1;
END_TRANSITION
STEP Oeffnen:
    SetSysActiv(N);
    I_Pumpe.M_A_FWD(N);
    I_Ventil_IN.M_A_OEFFNEN(N);
    I_Ventil_OUT.M_A_OEFFNEN(N);
    SetReady(N);
END_STEP
TRANSITION FROM Oeffnen TO Pumpen
    := I_Ventil_IN.P_Status = 1 AND I_Ventil_OUT.P_Status = 1 AND I_SekReady;
END_TRANSITION
STEP Pumpen:
    SetActiv(N);
    I_Pumpe.M_A_START(N);
END_STEP
TRANSITION FROM Pumpen TO Stoppen
    := NOT I_SekActiv AND I_Pumpe.P_Status = 2;
END_TRANSITION
STEP Stoppen:
    I_Pumpe.M_A_STOP(N);
END_STEP
TRANSITION FROM Stoppen TO Schliessen
    := I_Pumpe.P_Status = 1;
END_TRANSITION
STEP Schliessen:
    I_Ventil_IN.M_A_SCHLIESSEN(N);
    I_Ventil_OUT.M_A_SCHLIESSEN(N);
    ResetActiv(N);
END_STEP
TRANSITION FROM Schliessen TO Finished
    := I_Ventil_IN.P_Status = 0 AND I_Ventil_OUT.P_Status = 0;
END_TRANSITION
STEP Finished:
    ResetReady(N);
    M_Stop(N);
    ResetSysActiv(N);
END_STEP
TRANSITION FROM Finished TO Init
    := P_Status = 0;
END_TRANSITION

ACTION ResetActiv:
O_SW.ReactActiv:= FALSE;
O_SW.GF3Activ := FALSE;
END_ACTION

ACTION ResetReady:
O_SW.ReactReady := FALSE;
END_ACTION

ACTION ResetSysActiv:
GVL.SysState := 0;
END_ACTION

ACTION SetActiv:
O_SW.ReactActiv := TRUE;
O_SW.GF3Activ := TRUE;
END_ACTION

ACTION SetReady:
O_SW.ReactReady := TRUE;
END_ACTION

ACTION SetSysActiv:
GVL.SysState := 1;
END_ACTION

END_FUNCTION_BLOCK

// ---- POUs/03_Grundfuntkionen/GF_Ruehren.TcPOU
FUNCTION_BLOCK GF_Ruehren EXTENDS FB_Basis
VAR_INPUT
	// Instanzieren von Sensoren mit Interfaces
	
	// Instanzieren von Aktoren mit Interfaces
	I_Ruehrer		:I_Motor1R;
	// Rezeptparameter durch Controlword
	I_CW		:RezeptControlWord;	
END_VAR
VAR_OUTPUT
	O_SW		:RezeptStatusWord;
END_VAR
VAR
	
END_VAR

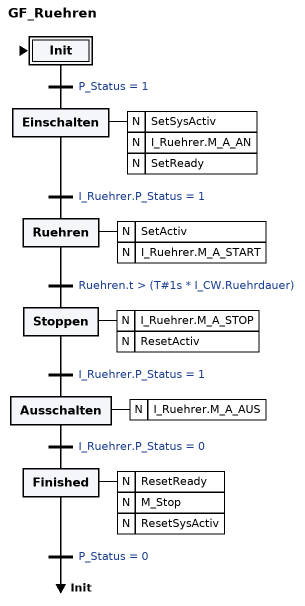
INITIAL_STEP Init:
END_STEP
TRANSITION FROM Init TO Einschalten
    := P_Status = 1;
END_TRANSITION
STEP Einschalten:
    SetSysActiv(N);
    I_Ruehrer.M_A_AN(N);
    SetReady(N);
END_STEP
TRANSITION FROM Einschalten TO Ruehren
    := I_Ruehrer.P_Status = 1;
END_TRANSITION
STEP Ruehren:
    SetActiv(N);
    I_Ruehrer.M_A_START(N);
END_STEP
TRANSITION FROM Ruehren TO Stoppen
    := Ruehren.t > (T#1s * I_CW.Ruehrdauer);
END_TRANSITION
STEP Stoppen:
    I_Ruehrer.M_A_STOP(N);
    ResetActiv(N);
END_STEP
TRANSITION FROM Stoppen TO Ausschalten
    := I_Ruehrer.P_Status = 1;
END_TRANSITION
STEP Ausschalten:
    I_Ruehrer.M_A_AUS(N);
END_STEP
TRANSITION FROM Ausschalten TO Finished
    := I_Ruehrer.P_Status = 0;
END_TRANSITION
STEP Finished:
    ResetReady(N);
    M_Stop(N);
    ResetSysActiv(N);
END_STEP
TRANSITION FROM Finished TO Init
    := P_Status = 0;
END_TRANSITION

ACTION ResetActiv:
O_SW.ReactActiv := FALSE;
O_SW.GF5Activ := FALSE;
END_ACTION

ACTION ResetReady:
O_SW.ReactReady := FALSE;
END_ACTION

ACTION ResetSysActiv:
GVL.SysState := 0;
END_ACTION

ACTION SetActiv:
O_SW.ReactActiv := TRUE;
O_SW.GF5Activ := TRUE;
END_ACTION

ACTION SetReady:
O_SW.ReactReady := TRUE;
END_ACTION

ACTION SetSysActiv:
GVL.SysState := 1;
END_ACTION

END_FUNCTION_BLOCK

// ---- POUs/03_Grundfuntkionen/GF_Warten.TcPOU
FUNCTION_BLOCK GF_Warten EXTENDS FB_Basis
VAR_INPUT
	// Instanzieren von Sensoren mit Interfaces
	
	// Instanzieren von Aktoren mit Interfaces
	
	// Rezeptparameter durch Controlword
	I_CW		:RezeptControlWord;	
END_VAR
VAR_OUTPUT
	O_SW		:RezeptStatusWord;
END_VAR
VAR
	
END_VAR

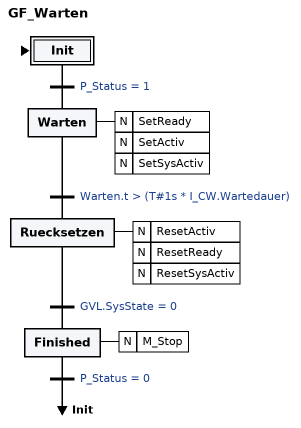
INITIAL_STEP Init:
END_STEP
TRANSITION FROM Init TO Warten
    := P_Status = 1;
END_TRANSITION
STEP Warten:
    SetReady(N);
    SetActiv(N);
    SetSysActiv(N);
END_STEP
TRANSITION FROM Warten TO Ruecksetzen
    := Warten.t > (T#1s * I_CW.Wartedauer);
END_TRANSITION
STEP Ruecksetzen:
    ResetActiv(N);
    ResetReady(N);
    ResetSysActiv(N);
END_STEP
TRANSITION FROM Ruecksetzen TO Finished
    := GVL.SysState = 0;
END_TRANSITION
STEP Finished:
    M_Stop(N);
END_STEP
TRANSITION FROM Finished TO Init
    := P_Status = 0;
END_TRANSITION

ACTION ResetActiv:
O_SW.ReactActiv := FALSE;
O_SW.GF6Activ := FALSE;
END_ACTION

ACTION ResetReady:
O_SW.ReactReady := FALSE;
END_ACTION

ACTION ResetSysActiv:
GVL.SysState := 0;
END_ACTION

ACTION SetActiv:
O_SW.ReactActiv := TRUE;
O_SW.GF6Activ := TRUE;
END_ACTION

ACTION SetReady:
O_SW.ReactReady := TRUE;
O_SW.SysReady := TRUE; 		// Damit auf oberen Stufen nicht auf 0 überschrieben wird
END_ACTION

ACTION SetSysActiv:
GVL.SysState := 1;
END_ACTION

END_FUNCTION_BLOCK

// ---- POUs/03_Grundfuntkionen/GF_Zirkulieren.TcPOU
FUNCTION_BLOCK GF_Zirkulieren EXTENDS FB_Basis
VAR_INPUT
	// Instanzieren von Sensoren mit Interfaces
	
	// Instanzieren von Aktoren mit Interfaces
	I_Ventil_IN			:I_Magnetventil;
	I_Ventil_OUT			:I_Magnetventil;
	
	I_Pumpe				:I_Motor2R;
	// Rezeptparameter durch Controlword
	I_CW		:RezeptControlWord;	
END_VAR

VAR_OUTPUT
	O_SW		:RezeptStatusWord;
END_VAR
VAR
	
END_VAR

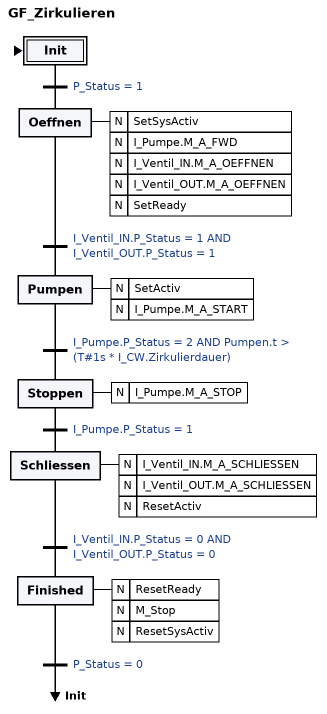
INITIAL_STEP Init:
END_STEP
TRANSITION FROM Init TO Oeffnen
    := P_Status = 1;
END_TRANSITION
STEP Oeffnen:
    SetSysActiv(N);
    I_Pumpe.M_A_FWD(N);
    I_Ventil_IN.M_A_OEFFNEN(N);
    I_Ventil_OUT.M_A_OEFFNEN(N);
    SetReady(N);
END_STEP
TRANSITION FROM Oeffnen TO Pumpen
    := I_Ventil_IN.P_Status = 1 AND I_Ventil_OUT.P_Status = 1;
END_TRANSITION
STEP Pumpen:
    SetActiv(N);
    I_Pumpe.M_A_START(N);
END_STEP
TRANSITION FROM Pumpen TO Stoppen
    := I_Pumpe.P_Status = 2 AND Pumpen.t > (T#1s * I_CW.Zirkulierdauer);
END_TRANSITION
STEP Stoppen:
    I_Pumpe.M_A_STOP(N);
END_STEP
TRANSITION FROM Stoppen TO Schliessen
    := I_Pumpe.P_Status = 1;
END_TRANSITION
STEP Schliessen:
    I_Ventil_IN.M_A_SCHLIESSEN(N);
    I_Ventil_OUT.M_A_SCHLIESSEN(N);
    ResetActiv(N);
END_STEP
TRANSITION FROM Schliessen TO Finished
    := I_Ventil_IN.P_Status = 0 AND I_Ventil_OUT.P_Status = 0;
END_TRANSITION
STEP Finished:
    ResetReady(N);
    M_Stop(N);
    ResetSysActiv(N);
END_STEP
TRANSITION FROM Finished TO Init
    := P_Status = 0;
END_TRANSITION

ACTION ResetActiv:
O_SW.ReactActiv := FALSE;
O_SW.GF8Activ := FALSE;
END_ACTION

ACTION ResetReady:
O_SW.ReactReady:= FALSE;
END_ACTION

ACTION ResetSysActiv:
GVL.SysState := 0;
END_ACTION

ACTION SetActiv:
O_SW.ReactActiv := TRUE;
O_SW.GF8Activ := TRUE;
END_ACTION

ACTION SetReady:
O_SW.ReactReady := TRUE;
END_ACTION

ACTION SetSysActiv:
GVL.SysState := 1;
END_ACTION

END_FUNCTION_BLOCK

// ---- GlobalTextList.TcGTLO
TEXTLIST GlobalTextList
  737 = '%f'
  656 = '%i'
  82 = '%s'
  520 = 'Auffüllprozess läuft'
  663 = 'AUTO'
  988 = 'Controll-Word'
  461 = 'Debug-HMI'
  776 = 'Definiert welche Leitung verwendet wird'
  578 = 'Definierte Temperatur für Heiz- / Kühlprozess'
  47 = 'Definierter sekundär-Reaktor'
  881 = 'Eigenschaften'
  587 = 'Eigenschaften & Inputs'
  668 = 'Enleermenge'
  20 = 'Entleerprozess läuft'
  350 = 'ERROR'
  1156 = 'Error'
  1154 = 'ERROR-ID'
  844 = 'ERROR-ID:'
  102 = 'ERROR:'
  771 = 'ERROR_ID'
  225 = 'FB_Füllstandsensor'
  379 = 'FB_HKSystem'
  89 = 'FB_Magnetventil'
  583 = 'FB_Motor1R'
  65 = 'FB_Motor2R'
  234 = 'FB_Temperatursensor'
  426 = 'Feldgerät-Steuerung'
  496 = 'Füllstandsensor'
  372 = 'GF1Activ'
  913 = 'GF2Activ'
  524 = 'GF3Activ'
  479 = 'GF4Activ'
  606 = 'GF5Activ'
  300 = 'GF6Activ'
  505 = 'GF7Activ'
  571 = 'GF8Activ'
  534 = 'Haltedauer'
  600 = 'Halteprozess läuft'
  705 = 'Heiz- / Kühlprozess läuft'
  42 = 'HK-System'
  333 = 'Input-Signal'
  828 = 'Input-Signal:'
  745 = 'Inputs'
  999 = 'I_iGeschw'
  510 = 'I_iSignal'
  254 = 'I_iTemp'
  916 = 'I_rHigh'
  121 = 'I_rLow'
  285 = 'I_rMax'
  680 = 'I_rMin'
  942 = 'Leitung'
  348 = 'MAN'
  975 = 'Messwert'
  1134 = 'Messwert:'
  64 = 'Methodenhandling'
  581 = 'MODI:'
  242 = 'Modus'
  278 = 'M_M_AN'
  0 = 'M_M_AUS'
  843 = 'M_M_BWD'
  38 = 'M_M_FWD'
  739 = 'M_M_HK_AN'
  330 = 'M_M_HK_AUS'
  478 = 'M_M_OEFFNEN'
  994 = 'M_M_PUMPE_AN'
  78 = 'M_M_PUMPE_AUS'
  727 = 'M_M_SCHLIESSEN'
  150 = 'M_M_START'
  41 = 'M_M_STOP'
  28 = 'Outputs '
  547 = 'O_bAktivieren'
  721 = 'O_bError'
  2 = 'O_bHeizen'
  342 = 'O_bKuehlen'
  866 = 'O_bPower'
  746 = 'O_bPumpen'
  544 = 'O_bRichtung'
  418 = 'O_iDrz'
  518 = 'O_iStoerungID'
  932 = 'POWER:'
  450 = 'PrimeActiv'
  282 = 'PrimReady'
  351 = 'Primärreaktor führt Prozess aus'
  770 = 'Primärreaktor ist bereit für den Prozess'
  331 = 'Pumpe'
  722 = 'Pumpmenge'
  152 = 'Pumpprozess läuft'
  1029 = 'P_DefTemp:'
  685 = 'P_GrenzeOben'
  502 = 'P_GrenzeUnten'
  794 = 'P_Laufzeit'
  293 = 'P_MaxDrz'
  323 = 'P_MaxDrz:'
  692 = 'P_Messwert'
  758 = 'P_Zustand'
  545 = 'Remperatursensor'
  503 = 'Reset'
  954 = 'RESET:'
  946 = 'Ruehrdauer'
  933 = 'Rührer'
  40 = 'Rührprozess läuft'
  616 = 'SekActiv'
  650 = 'SekReady'
  373 = 'SekReakt'
  560 = 'Sekundärreaktor führt Prozess aus'
  923 = 'Sekundärreaktor ist bereit für den Prozess'
  860 = 'Start'
  857 = 'Start sekundär Reaktor'
  979 = 'Status-Word'
  973 = 'Temp'
  27 = 'Temperatursensor'
  993 = 'Verbunden'
  217 = 'VERBUNDEN'
  834 = 'VERBUNDEN:'
  90 = 'VERRIEGELN:'
  889 = 'Wartedauer'
  362 = 'Warteprozess läuft'
  438 = 'Wie lange soll gerührt werden'
  301 = 'Wie lange soll gerührt werden '
  246 = 'Wie lange soll TEmperatur gehalten werden'
  394 = 'Wie lange soll Temperatur gehalten werden'
  666 = 'Wie lange soll zirkuliert werden'
  768 = 'Zierkulierdauer'
  926 = 'Zirkulierprozess läuft'
  26 = 'Zu entleerende Menge'
  164 = 'Zu pumpende Menge'
END_TEXTLIST
